INTERFACE I_SafetyBase EXTENDS I_Component, I_Resettable, I_SafetySimulation, I_TaskResult

{attribute 'monitoring' := 'call'}
PROPERTY OK : BOOL
GET
END_GET
END_PROPERTY

PROPERTY ResetFunction : I_SafetyReset
SET
END_SET
END_PROPERTY

END_INTERFACE

(* stored: Version 1.1.0.1, ProductVersion 3.1.4026.18
   Itf I_SafetyBase: Id {33cdca74-ea3a-06f2-0eb4-beaa47fde1de}
   Property OK: Id {e0b95048-8d34-0742-1bc2-2e478b2bf63f}
   Get Get: Id {1b196e97-c4df-0d05-36fe-37a5f988eac4}
   Property ResetFunction: Id {c1ee9de6-a76e-47a1-b1dc-9c3695e49a5b}
   Set Set: Id {77bda360-72a9-4a6a-b0b0-d54c26cc427e} *)
